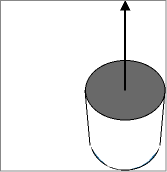
VISUALIZATION VISU_Tube_Top_4  // 167x172
VAR_IN_OUT
	azi : LREAL;
END_VAR
    Ellipse (90,110 70x60)
        p2858320360: azi
    Polygon (85,90) (165,90) (160,145) (160,145) (156,152) (153,155) (148,161) (140,166) (130,169) (118,169) (108,166) (100,159) (95,153) (90,145)
        p2858320360: azi
    Ellipse (85,60 80x60)
        p2858320360: azi
    Polygon (120,10) (125,0) (130,10)
        p2858320360: azi
    Polyline (125,90) (125,10)
        p2858320360: azi
    Polyline (90,145) (85,90)
        p2858320360: azi
    Polyline (160,145) (165,90)
        p2858320360: azi
END_VISUALIZATION

(* stored: Version 1.1.0.1, ProductVersion 3.1.4018.5
   Visu VISU_Tube_Top_4: Id {3d477afb-ee98-4397-95b4-d86cc44a7969} *)
